(* IEC 61131-3 sources: CodeSys/, 2 files *)

(* ---- ST_code.st ---- *)
// into the upper window in CodeSys:
PROGRAM PLC_PRG
VAR
	ixStart: BOOL;
	ixStop: BOOL;
	qxKM1: BOOL;
	mwMyInt: INT;
END_VAR

// into the lower window in CodeSys:
qxKM1:= (ixStart OR qxKM1) AND NOT ixStop;

IF qxKM1 = TRUE THEN
	mwMyInt:= mwMyInt + 1;
END_IF

(* ---- ST_generator(TON).st ---- *)
// into the upper window in CodeSys:
PROGRAM PLC_PRG
VAR
	xEnable0: BOOL;
	tMyTime: TIME;
	xPulse0: BOOL;
	MyTON0: TON;
	xGen1s: BOOL;
	xWork0: BOOL;
END_VAR

// into the lower window in CodeSys:
xWork0 := xEnable0 AND NOT xPulse0;
MyTON0 (IN := xWork0, PT := T#1S);
xPulse0 := MyTON0.Q;
tMyTime := MyTON0.ET;
xGen1s := (tMyTime <= T#500MS);
